{attribute 'qualified_only'}
{attribute 'strict'}
TYPE E_CRYO_CPA_DIAG_IDX :
(
	WATER_IN	:= 0,
	WATER_OUT,
	OIL_TEMP,
	HELIUM_TEMP,
	HELIUM_LOW_PRESS_OP,
	HELIUM_HIGH_PRESS_OP,
	HELIUM_DELTA_PRESS,
	HELIUM_STATIC_LOW_PRESS,
	HELIUM_STATIC_HIGH_PRESS
);
END_TYPE

(* stored: Version 1.1.0.1, ProductVersion 3.1.4024.9
   DUT E_CRYO_CPA_DIAG_IDX: Id {745f7abf-cf3c-43ae-a948-93b1e24664cb} *)
